Omron CX-Programmer project NuovoProgetto (CX-Programmer 8.01)

# PLC PLC: CJ1M CPU23

## Global symbols (name address type ; comment)
A W5 INT  ; PER AZZERAMENTO VARIABILI
A0.01 BOOL  ; 0.2
CICLO W0.00 BOOL[15]
CancelloAutomatico cancello_automatico
ControlloLivello controllo_livello
ENABLE W0.15 BOOL
GARAGE garage
IN00 0.00 BOOL  ; IN00
IN01 0.01 BOOL  ; IN01
IN02 0.02 BOOL  ; IN02
IN03 0.03 BOOL  ; IN03
IN04 0.04 BOOL  ; IN04
IN05 0.05 BOOL  ; IN05
IN06 0.06 BOOL  ; IN06
IN07 0.07 BOOL  ; IN07
IN08 0.08 BOOL  ; IN08
IN09 0.09 BOOL  ; IN09
IN10 0.10 BOOL  ; IN10
IN11 0.11 BOOL  ; IN11
IN12 0.12 BOOL  ; IN12
IN13 0.13 BOOL  ; IN13
IN14 0.14 BOOL  ; IN14
IN15 0.15 BOOL  ; IN15
IN16 1.00 BOOL  ; IN16
MAT2 inversione_di_marcia_MAT
MAT3 stella_triangolo_MAT
MarciaArresto marcia_arresto_MAT
Miscelatore miscelatore
OLD_OPZIONE W10 INT
OPZIONE W15 INT  ; SCELTA DEL CICLO
OUT00 2.00 BOOL  ; OUT00
OUT01 2.01 BOOL  ; OUT01
OUT02 2.02 BOOL  ; OUT02
OUT03 2.03 BOOL  ; OUT03
OUT04 2.04 BOOL  ; OUT04
OUT05 2.05 BOOL  ; OUT05
OUT06 2.06 BOOL  ; OUT06
OUT07 2.07 BOOL  ; OUT07
OUT08 2.08 BOOL  ; OUT08
OUT09 2.09 BOOL  ; OUT09
OUT10 2.10 BOOL  ; OUT10
OUT11 2.11 BOOL  ; OUT11
OUT12 2.12 BOOL  ; OUT12
OUT13 2.13 BOOL  ; OUT13
OUT14 2.14 BOOL  ; OUT14
OUT15 2.15 BOOL  ; OUT15
OUTCOUNTER1 D60 INT  ; uscita visione counter1
OUTCOUNTER2 D70 INT  ; uscita visione counter2
OUTCOUNTER3 D80 INT  ; uscita visione counter3
OUTCOUNTER4 D90 INT  ; uscita visione counter4
OUTCOUNTER5 D100 INT  ; uscita visione counter5
OUTCOUNTER6 D110 INT  ; uscita visione counter6
OUTTIMER1 D0 INT  ; uscita visione timer1
OUTTIMER2 D10 INT  ; uscita visione timer2
OUTTIMER3 D20 INT  ; uscita visione timer3
OUTTIMER4 D30 INT  ; uscita visione timer4
OUTTIMER5 D40 INT  ; uscita visione timer5
OUTTIMER6 D50 INT  ; uscita visione timer6
START 0.08 BOOL  ; INStart
SemaforoPedonale semaforo_pedonale
elp2 ciclo_elettropneumatico_due
elp3 ciclo_elettropneumatico_tre_mono
pos3 ciclo_elettropneumatico_uno

## Program CICLO_AVVIO (cyclic task 0)
; CICLO DI PARTENZA CON LA DEFINIZIONE DI TUTTI I BLOCCHI
Local symbols
RESET W100.02 BOOL
TERM1 W100.00 BOOL
TERM2 W100.01 BOOL

### Section RICHIAMMO_BLOCCHI

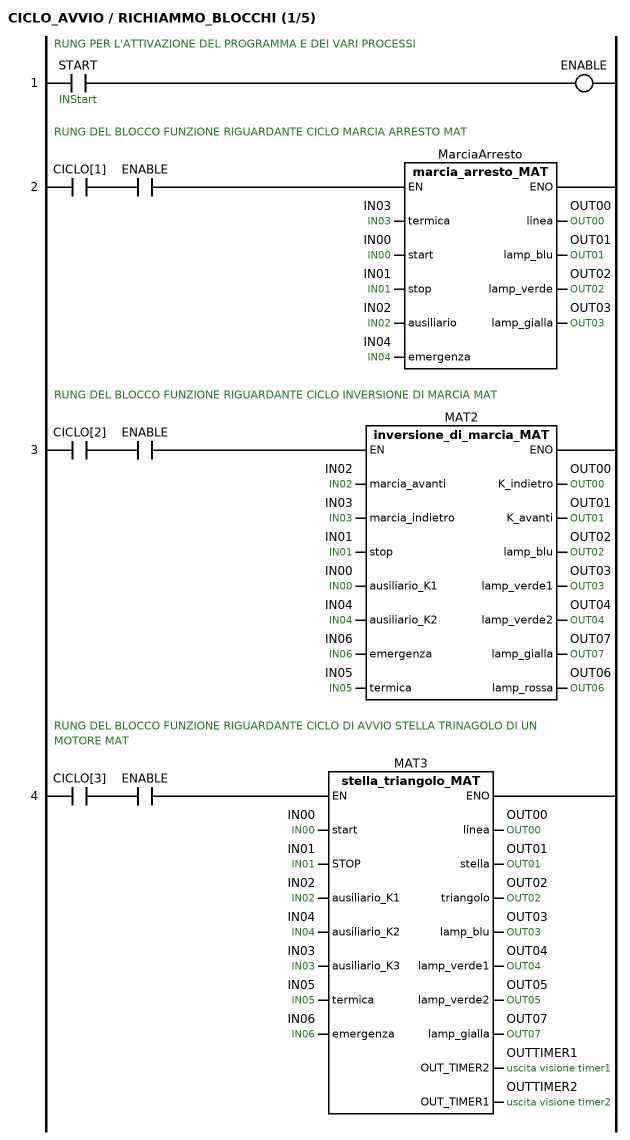
; rung 1: RUNG PER L'ATTIVAZIONE DEL PROGRAMMA E DEI VARI PROCESSI
LD START  ; INStart
OUT ENABLE
; rung 2: RUNG DEL BLOCCO FUNZIONE RIGUARDANTE CICLO MARCIA ARRESTO MAT
LD CICLO[1]
AND ENABLE
CALL MarciaArresto : marcia_arresto_MAT (termica := IN03, start := IN00, stop := IN01, ausiliario := IN02, emergenza := IN04, linea => OUT00, lamp_blu => OUT01, lamp_verde => OUT02, lamp_gialla => OUT03)  ; IN03, IN00, IN01, IN02, IN04, OUT00, OUT01, OUT02, OUT03
; rung 3: RUNG DEL BLOCCO FUNZIONE RIGUARDANTE CICLO INVERSIONE DI MARCIA MAT
LD CICLO[2]
AND ENABLE
CALL MAT2 : inversione_di_marcia_MAT (marcia_avanti := IN02, marcia_indietro := IN03, stop := IN01, ausiliario_K1 := IN00, ausiliario_K2 := IN04, emergenza := IN06, termica := IN05, K_indietro => OUT00, K_avanti => OUT01, lamp_blu => OUT02, lamp_verde1 => OUT03, lamp_verde2 => OUT04, lamp_gialla => OUT07, lamp_rossa => OUT06)  ; IN02, IN03, IN01, IN00, IN04, IN06, IN05, OUT00, OUT01, OUT02, OUT03, OUT04, OUT07, OUT06
; rung 4: RUNG DEL BLOCCO FUNZIONE RIGUARDANTE CICLO DI AVVIO STELLA TRINAGOLO DI UN MOTORE MAT
LD CICLO[3]
AND ENABLE
CALL MAT3 : stella_triangolo_MAT (start := IN00, STOP := IN01, ausiliario_K1 := IN02, ausiliario_K2 := IN04, ausiliario_K3 := IN03, termica := IN05, emergenza := IN06, linea => OUT00, stella => OUT01, triangolo => OUT02, lamp_blu => OUT03, lamp_verde1 => OUT04, lamp_verde2 => OUT05, lamp_gialla => OUT07, OUT_TIMER2 => OUTTIMER1, OUT_TIMER1 => OUTTIMER2)  ; IN00, IN01, IN02, IN04, IN03, IN05, IN06, OUT00, OUT01, OUT02, OUT03, OUT04, OUT05, OUT07, uscita visione timer1, uscita visione timer2

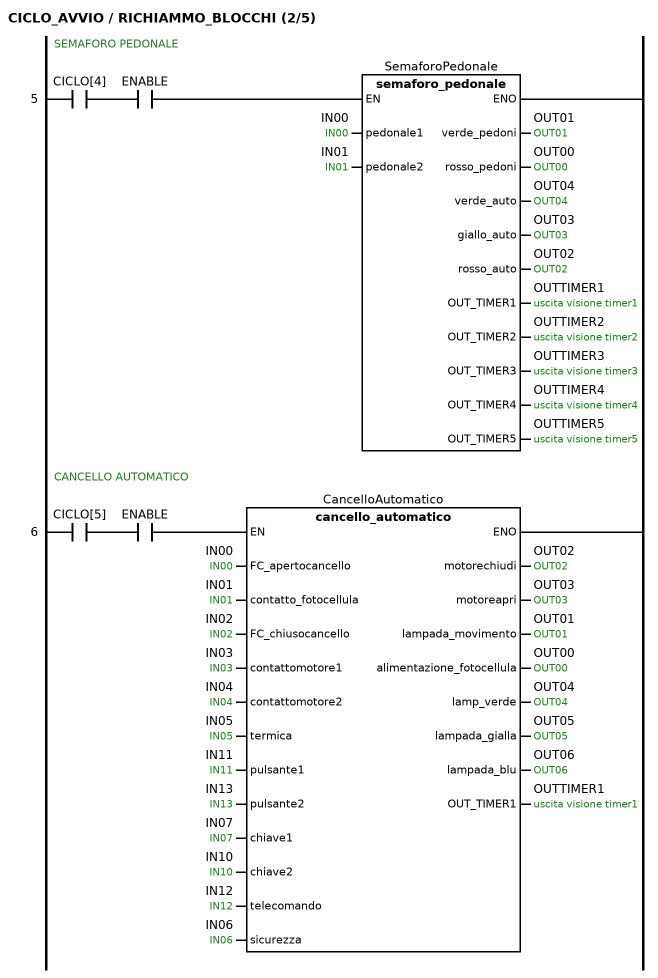
; rung 5: SEMAFORO PEDONALE
LD CICLO[4]
AND ENABLE
CALL SemaforoPedonale : semaforo_pedonale (pedonale1 := IN00, pedonale2 := IN01, verde_pedoni => OUT01, rosso_pedoni => OUT00, verde_auto => OUT04, giallo_auto => OUT03, rosso_auto => OUT02, OUT_TIMER1 => OUTTIMER1, OUT_TIMER2 => OUTTIMER2, OUT_TIMER3 => OUTTIMER3, OUT_TIMER4 => OUTTIMER4, OUT_TIMER5 => OUTTIMER5)  ; IN00, IN01, OUT01, OUT00, OUT04, OUT03, OUT02, uscita visione timer1, uscita visione timer2, uscita visione timer3, uscita visione timer4, uscita visione timer5
; rung 6: CANCELLO AUTOMATICO
LD CICLO[5]
AND ENABLE
CALL CancelloAutomatico : cancello_automatico (FC_apertocancello := IN00, contatto_fotocellula := IN01, FC_chiusocancello := IN02, contattomotore1 := IN03, contattomotore2 := IN04, termica := IN05, pulsante1 := IN11, pulsante2 := IN13, chiave1 := IN07, chiave2 := IN10, telecomando := IN12, sicurezza := IN06, motorechiudi => OUT02, motoreapri => OUT03, lampada_movimento => OUT01, alimentazione_fotocellula => OUT00, lamp_verde => OUT04, lampada_gialla => OUT05, lampada_blu => OUT06, OUT_TIMER1 => OUTTIMER1)  ; IN00, IN01, IN02, IN03, IN04, IN05, IN11, IN13, IN07, IN10, IN12, IN06, OUT02, OUT03, OUT01, OUT00, OUT04, OUT05, OUT06, uscita visione timer1

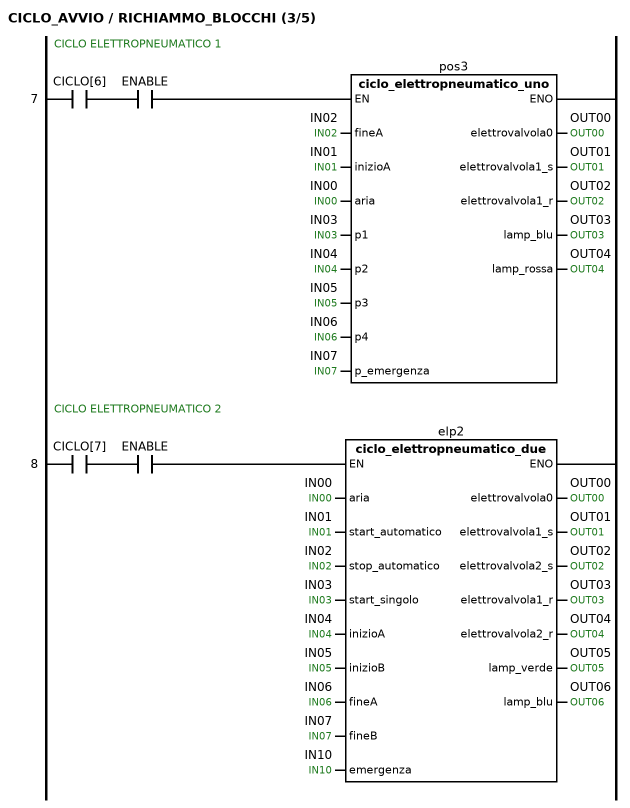
; rung 7: CICLO ELETTROPNEUMATICO 1
LD CICLO[6]
AND ENABLE
CALL pos3 : ciclo_elettropneumatico_uno (fineA := IN02, inizioA := IN01, aria := IN00, p1 := IN03, p2 := IN04, p3 := IN05, p4 := IN06, p_emergenza := IN07, elettrovalvola0 => OUT00, elettrovalvola1_s => OUT01, elettrovalvola1_r => OUT02, lamp_blu => OUT03, lamp_rossa => OUT04)  ; IN02, IN01, IN00, IN03, IN04, IN05, IN06, IN07, OUT00, OUT01, OUT02, OUT03, OUT04
; rung 8: CICLO ELETTROPNEUMATICO 2
LD CICLO[7]
AND ENABLE
CALL elp2 : ciclo_elettropneumatico_due (aria := IN00, start_automatico := IN01, stop_automatico := IN02, start_singolo := IN03, inizioA := IN04, inizioB := IN05, fineA := IN06, fineB := IN07, emergenza := IN10, elettrovalvola0 => OUT00, elettrovalvola1_s => OUT01, elettrovalvola2_s => OUT02, elettrovalvola1_r => OUT03, elettrovalvola2_r => OUT04, lamp_verde => OUT05, lamp_blu => OUT06)  ; IN00, IN01, IN02, IN03, IN04, IN05, IN06, IN07, IN10, OUT00, OUT01, OUT02, OUT03, OUT04, OUT05, OUT06

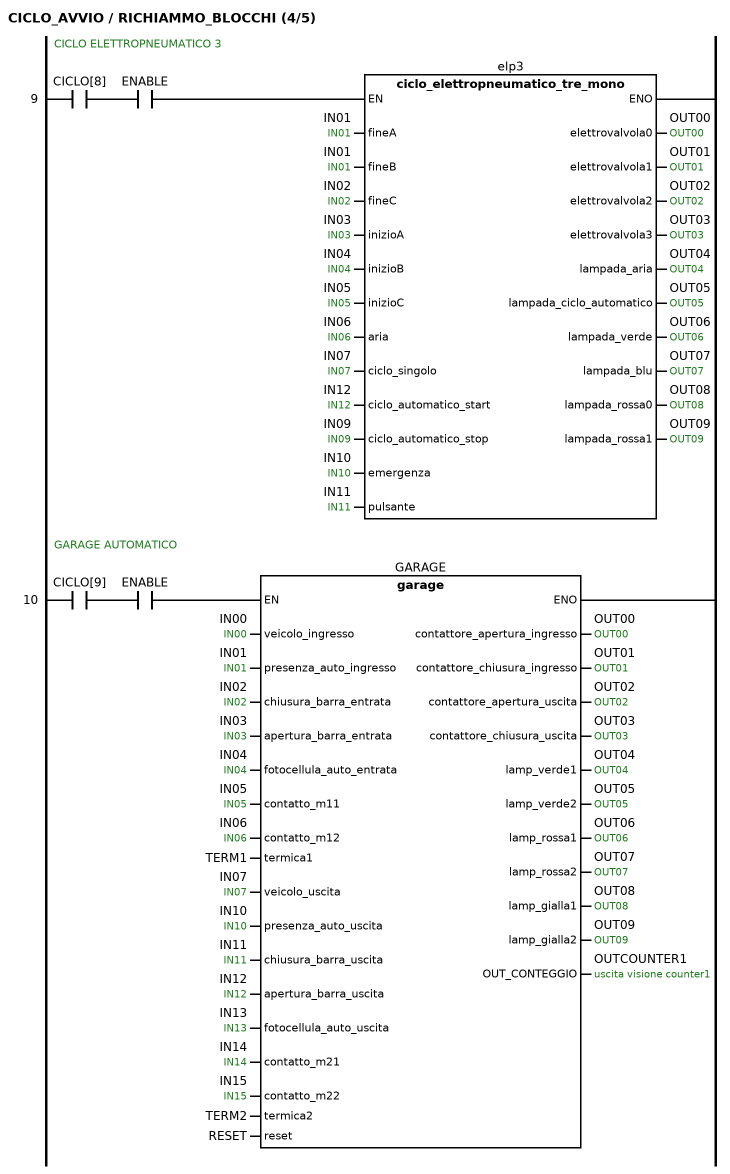
; rung 9: CICLO ELETTROPNEUMATICO 3
LD CICLO[8]
AND ENABLE
CALL elp3 : ciclo_elettropneumatico_tre_mono (fineA := IN01, fineB := IN01, fineC := IN02, inizioA := IN03, inizioB := IN04, inizioC := IN05, aria := IN06, ciclo_singolo := IN07, ciclo_automatico_start := IN12, ciclo_automatico_stop := IN09, emergenza := IN10, pulsante := IN11, elettrovalvola0 => OUT00, elettrovalvola1 => OUT01, elettrovalvola2 => OUT02, elettrovalvola3 => OUT03, lampada_aria => OUT04, lampada_ciclo_automatico => OUT05, lampada_verde => OUT06, lampada_blu => OUT07, lampada_rossa0 => OUT08, lampada_rossa1 => OUT09)  ; IN01, IN02, IN03, IN04, IN05, IN06, IN07, IN12, IN09, IN10, IN11, OUT00, OUT01, OUT02, OUT03, OUT04, OUT05, OUT06, OUT07, OUT08, OUT09
; rung 10: GARAGE AUTOMATICO
LD CICLO[9]
AND ENABLE
CALL GARAGE : garage (veicolo_ingresso := IN00, presenza_auto_ingresso := IN01, chiusura_barra_entrata := IN02, apertura_barra_entrata := IN03, fotocellula_auto_entrata := IN04, contatto_m11 := IN05, contatto_m12 := IN06, termica1 := TERM1, veicolo_uscita := IN07, presenza_auto_uscita := IN10, chiusura_barra_uscita := IN11, apertura_barra_uscita := IN12, fotocellula_auto_uscita := IN13, contatto_m21 := IN14, contatto_m22 := IN15, termica2 := TERM2, reset := RESET, contattore_apertura_ingresso => OUT00, contattore_chiusura_ingresso => OUT01, contattore_apertura_uscita => OUT02, contattore_chiusura_uscita => OUT03, lamp_verde1 => OUT04, lamp_verde2 => OUT05, lamp_rossa1 => OUT06, lamp_rossa2 => OUT07, lamp_gialla1 => OUT08, lamp_gialla2 => OUT09, OUT_CONTEGGIO => OUTCOUNTER1)  ; IN00, IN01, IN02, IN03, IN04, IN05, IN06, IN07, IN10, IN11, IN12, IN13, IN14, IN15, OUT00, OUT01, OUT02, OUT03, OUT04, OUT05, OUT06, OUT07, OUT08, OUT09, uscita visione counter1

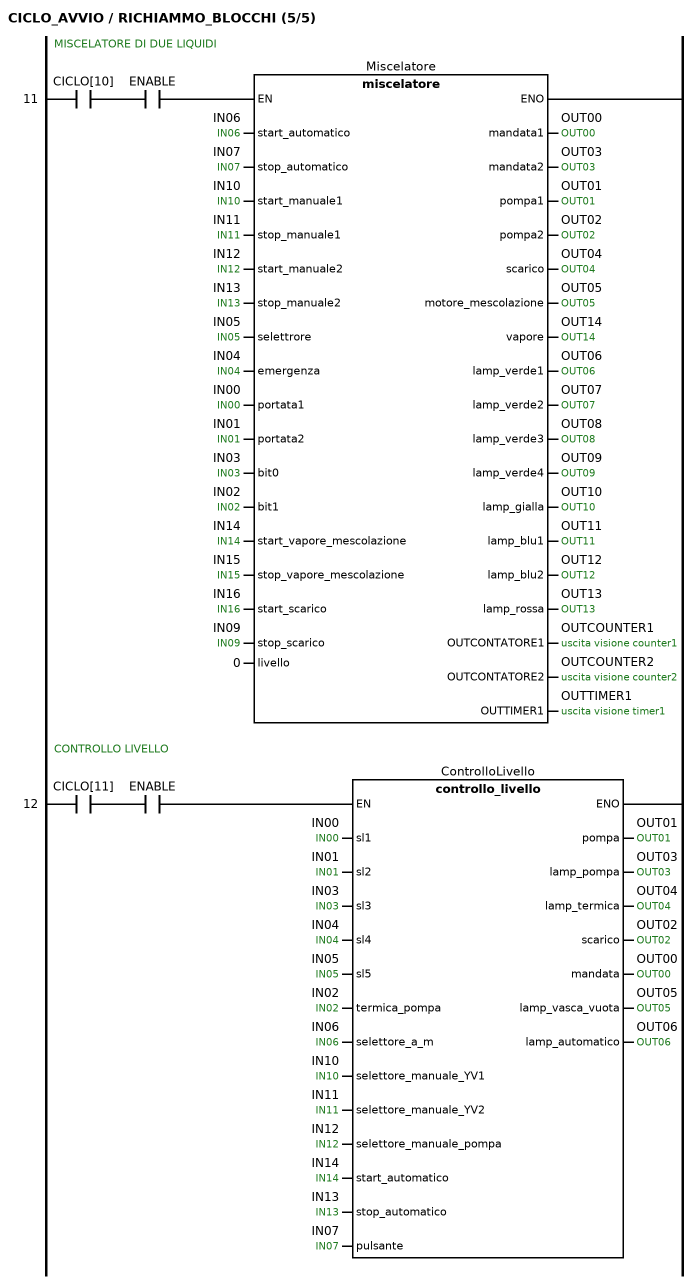
; rung 11: MISCELATORE DI DUE LIQUIDI
LD CICLO[10]
AND ENABLE
CALL Miscelatore : miscelatore (start_automatico := IN06, stop_automatico := IN07, start_manuale1 := IN10, stop_manuale1 := IN11, start_manuale2 := IN12, stop_manuale2 := IN13, selettrore := IN05, emergenza := IN04, portata1 := IN00, portata2 := IN01, bit0 := IN03, bit1 := IN02, start_vapore_mescolazione := IN14, stop_vapore_mescolazione := IN15, start_scarico := IN16, stop_scarico := IN09, livello := 0, mandata1 => OUT00, mandata2 => OUT03, pompa1 => OUT01, pompa2 => OUT02, scarico => OUT04, motore_mescolazione => OUT05, vapore => OUT14, lamp_verde1 => OUT06, lamp_verde2 => OUT07, lamp_verde3 => OUT08, lamp_verde4 => OUT09, lamp_gialla => OUT10, lamp_blu1 => OUT11, lamp_blu2 => OUT12, lamp_rossa => OUT13, OUTCONTATORE1 => OUTCOUNTER1, OUTCONTATORE2 => OUTCOUNTER2, OUTTIMER1 => OUTTIMER1)  ; IN06, IN07, IN10, IN11, IN12, IN13, IN05, IN04, IN00, IN01, IN03, IN02, IN14, IN15, IN16, IN09, OUT00, OUT03, OUT01, OUT02, OUT04, OUT05, OUT14, OUT06, OUT07, OUT08, OUT09, OUT10, OUT11, OUT12, OUT13, uscita visione counter1, uscita visione counter2, uscita visione timer1
; rung 12: CONTROLLO LIVELLO
LD CICLO[11]
AND ENABLE
CALL ControlloLivello : controllo_livello (sl1 := IN00, sl2 := IN01, sl3 := IN03, sl4 := IN04, sl5 := IN05, termica_pompa := IN02, selettore_a_m := IN06, selettore_manuale_YV1 := IN10, selettore_manuale_YV2 := IN11, selettore_manuale_pompa := IN12, start_automatico := IN14, stop_automatico := IN13, pulsante := IN07, pompa => OUT01, lamp_pompa => OUT03, lamp_termica => OUT04, scarico => OUT02, mandata => OUT00, lamp_vasca_vuota => OUT05, lamp_automatico => OUT06)  ; IN00, IN01, IN03, IN04, IN05, IN02, IN06, IN10, IN11, IN12, IN14, IN13, IN07, OUT01, OUT03, OUT04, OUT02, OUT00, OUT05, OUT06

### Section END
; rung 0
END(001)

## Program SCELTA (cyclic task 1)
; SCELTA
(*DOPO AVER RICEVUTO IL VALORE DI POSIZIONE SI ESEGUE LA VERIFICA COMPARANDO I VALORI PRECENTI  
CON QUELLI ATTUALI:
-SE CORRISPONDONO TUTTO OK  
-SE  DIVERSI VENGONO AGGIORNATI AI VALORI ATTUALI ( CICLO[] ) 
SUCCESSIVAMENTE MODIFICANO GLI ENABLE DEI BLOCCHI*)
IF ENABLE THEN
	
	IF OPZIONE =  OLD_OPZIONE THEN  		(* SE LA VARIABILE OPZIONE NON E' CAMBIATA NON ESEGUO NIENTE *)
	
			OLD_OPZIONE := OPZIONE;	
			
	ELSE
			(* AZZERAMENTO USCITE NEL CAMBIO DI STATO*)
			OUT00 := FALSE;
			OUT01 := FALSE;
			OUT02 := FALSE;
			OUT03 := FALSE;
			OUT04 := FALSE;
			OUT05 := FALSE;
			OUT06 := FALSE;
			OUT07 := FALSE;
			OUT08 := FALSE;
			OUT09 := FALSE;
			OUT10 := FALSE;
			OUT11 := FALSE;
			OUT12 := FALSE;
			OUT13 := FALSE;
			OUT14 := FALSE;
			OUT15:= FALSE;
			
			(* AZZERAMENTO USCITE NEL CAMBIO DI STATO*)			
			IN00 := FALSE;
			IN01 := FALSE;
			IN02 := FALSE;
			IN03 := FALSE;
			IN04 := FALSE;
			IN05 := FALSE;
			IN06 := FALSE;
			IN07 := FALSE;
			IN10 := FALSE;
			IN11 := FALSE;
			IN12 := FALSE;
			IN13 := FALSE;
			IN14 := FALSE;
			IN15:= FALSE;
			IN16 := FALSE;
				
                        (*SE LA VARIABILE OPZIONE E' CAMBIATA SI VERIFICA IL VALORE E SI CAMBIA IL BIT CORRISPONDENTE *)
			FOR A := 1 TO 11 BY 1 DO			(*CICLO PER ANDARE A CAMBIARE I VALORI DEI BIT*)

				IF A = OPZIONE  THEN            		(*CONFRONTO TRA INDICE E POSIZIONE*)
			
					CICLO[OPZIONE] := TRUE; 	(*SE IL VALORE E' UGUALE METTO A 1 IL BIT *)  
			
				ELSE
			
					CICLO[A] := FALSE; 		(*SE IL VALORE E' DIVERSO METTO A 0 IL BIT *)
			
				END_IF;
			
			END_FOR	;
	
	OLD_OPZIONE := OPZIONE; 			(*AGGIORNO IL VALORE DI OLD_OPZIONE*)

	END_IF;		

END_IF;;

## Function block cancello_automatico
VAR_INPUT
  FC_apertocancello : BOOL;
  contatto_fotocellula : BOOL;
  FC_chiusocancello : BOOL;
  contattomotore1 : BOOL;
  contattomotore2 : BOOL;
  termica : BOOL;
  pulsante1 : BOOL;
  pulsante2 : BOOL;
  chiave1 : BOOL;
  chiave2 : BOOL;
  telecomando : BOOL;
  sicurezza : BOOL;
END_VAR
VAR_OUTPUT
  motorechiudi : BOOL;
  motoreapri : BOOL;
  lampada_movimento : BOOL;
  alimentazione_fotocellula : BOOL;
  lamp_verde : BOOL;
  lampada_gialla : BOOL;
  lampada_blu : BOOL;
  OUT_TIMER1 : INT;
END_VAR
VAR
  MEM1 : BOOL;
  MEM2 : BOOL;
  MEM3 : BOOL;
  TIME1 : TIMER;
END_VAR

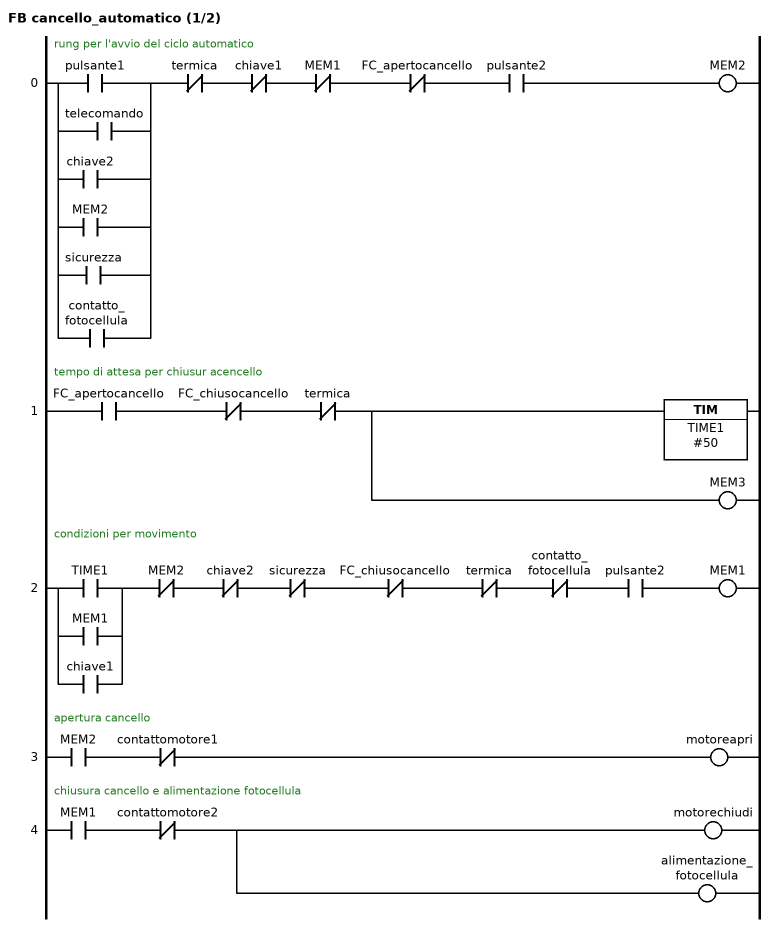
; rung 0: rung per l'avvio del ciclo automatico
LD pulsante1
OR telecomando
OR chiave2
OR MEM2
OR sicurezza
OR contatto_fotocellula
ANDNOT termica
ANDNOT chiave1
ANDNOT MEM1
ANDNOT FC_apertocancello
AND pulsante2
OUT MEM2
; rung 1: tempo di attesa per chiusur acencello
LD FC_apertocancello
ANDNOT FC_chiusocancello
ANDNOT termica
TIM TIME1 #50
OUT MEM3
; rung 2: condizioni per movimento
LD TIME1
OR MEM1
OR chiave1
ANDNOT MEM2
ANDNOT chiave2
ANDNOT sicurezza
ANDNOT FC_chiusocancello
ANDNOT termica
ANDNOT contatto_fotocellula
AND pulsante2
OUT MEM1
; rung 3: apertura cancello
LD MEM2
ANDNOT contattomotore1
OUT motoreapri
; rung 4: chiusura cancello e alimentazione fotocellula
LD MEM1
ANDNOT contattomotore2
OUT motorechiudi
OUT alimentazione_fotocellula

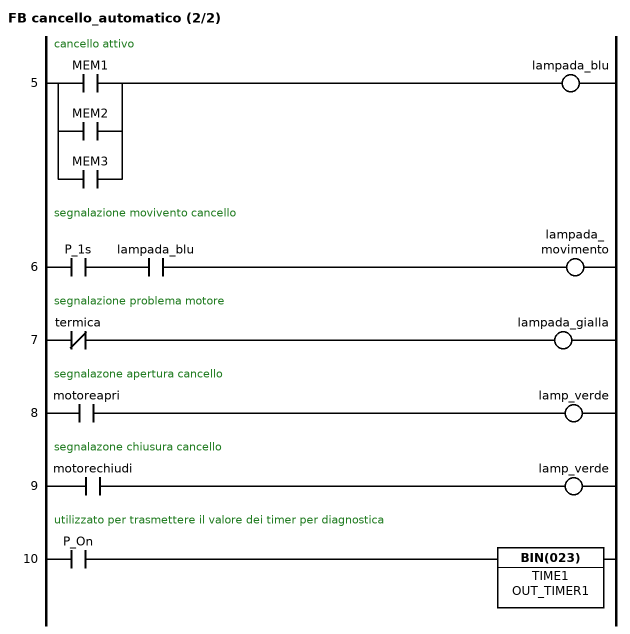
; rung 5: cancello attivo
LD MEM1
OR MEM2
OR MEM3
OUT lampada_blu
; rung 6: segnalazione movivento cancello
LD P_1s
AND lampada_blu
OUT lampada_movimento
; rung 7: segnalazione problema motore
LDNOT termica
OUT lampada_gialla
; rung 8: segnalazone apertura cancello
LD motoreapri
OUT lamp_verde
; rung 9: segnalazone chiusura cancello
LD motorechiudi
OUT lamp_verde
; rung 10: utilizzato per trasmettere il valore dei timer per diagnostica
LD P_On
BIN(023) TIME1 OUT_TIMER1

## Function block ciclo_elettropneumatico_due
VAR_INPUT
  aria : BOOL;
  start_automatico : BOOL;
  stop_automatico : BOOL;
  start_singolo : BOOL;
  inizioA : BOOL;
  inizioB : BOOL;
  fineA : BOOL;
  fineB : BOOL;
  emergenza : BOOL;
END_VAR
VAR_OUTPUT
  elettrovalvola0 : BOOL;
  elettrovalvola1_s : BOOL;
  elettrovalvola2_s : BOOL;
  elettrovalvola1_r : BOOL;
  elettrovalvola2_r : BOOL;
  lamp_verde : BOOL;
  lamp_blu : BOOL;
END_VAR
VAR
  MEM2 : BOOL;
  MEM1 : BOOL;
END_VAR

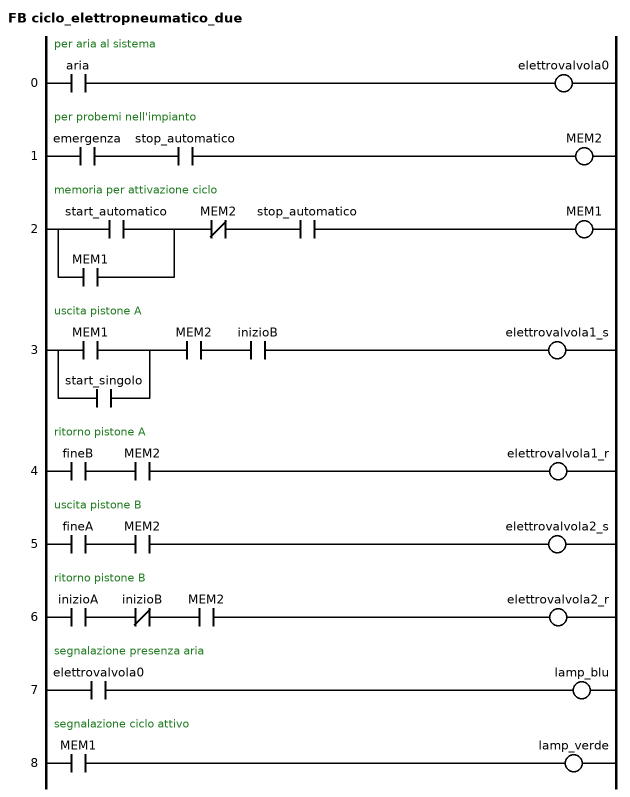
; rung 0: per aria al sistema
LD aria
OUT elettrovalvola0
; rung 1: per probemi nell'impianto
LD emergenza
AND stop_automatico
OUT MEM2
; rung 2: memoria per attivazione ciclo
LD start_automatico
OR MEM1
ANDNOT MEM2
AND stop_automatico
OUT MEM1
; rung 3: uscita pistone A
LD MEM1
OR start_singolo
AND MEM2
AND inizioB
OUT elettrovalvola1_s
; rung 4: ritorno pistone A
LD fineB
AND MEM2
OUT elettrovalvola1_r
; rung 5: uscita pistone B
LD fineA
AND MEM2
OUT elettrovalvola2_s
; rung 6: ritorno pistone B
LD inizioA
ANDNOT inizioB
AND MEM2
OUT elettrovalvola2_r
; rung 7: segnalazione presenza aria
LD elettrovalvola0
OUT lamp_blu
; rung 8: segnalazione ciclo attivo
LD MEM1
OUT lamp_verde

## Function block ciclo_elettropneumatico_tre_mono
VAR_INPUT
  fineA : BOOL;
  fineB : BOOL;
  fineC : BOOL;
  inizioA : BOOL;
  inizioB : BOOL;
  inizioC : BOOL;
  aria : BOOL;
  ciclo_singolo : BOOL;
  ciclo_automatico_start : BOOL;
  ciclo_automatico_stop : BOOL;
  emergenza : BOOL;
  pulsante : BOOL;
END_VAR
VAR_OUTPUT
  elettrovalvola0 : BOOL;
  elettrovalvola1 : BOOL;
  elettrovalvola2 : BOOL;
  elettrovalvola3 : BOOL;
  lampada_aria : BOOL;
  lampada_ciclo_automatico : BOOL;
  lampada_verde : BOOL;
  lampada_blu : BOOL;
  lampada_rossa0 : BOOL;
  lampada_rossa1 : BOOL;
END_VAR
VAR
  MEM1 : BOOL;
  MEM2 : BOOL;
END_VAR

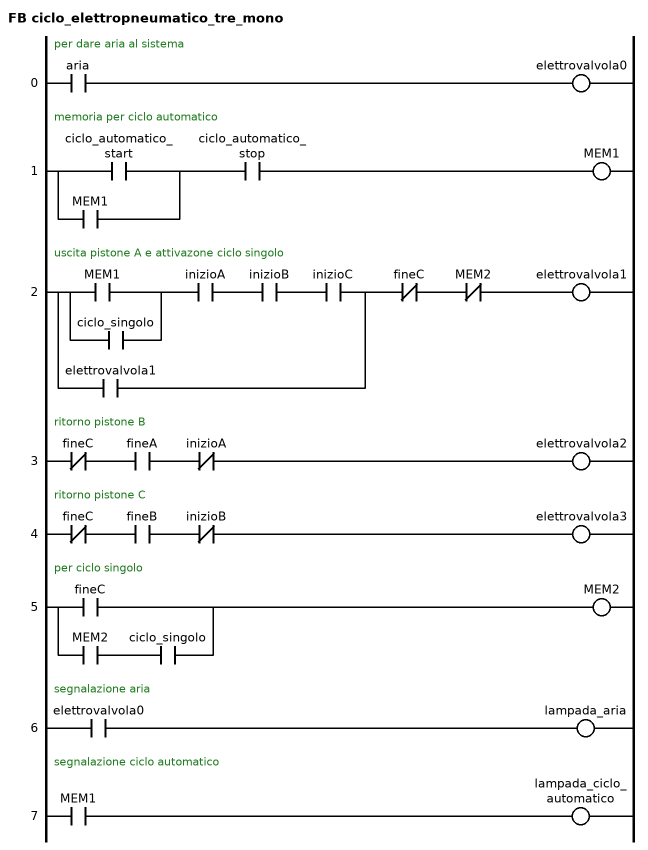
; rung 0: per dare aria al sistema
LD aria
OUT elettrovalvola0
; rung 1: memoria per ciclo automatico
LD ciclo_automatico_start
OR MEM1
AND ciclo_automatico_stop
OUT MEM1
; rung 2: uscita pistone A e attivazone ciclo singolo
LD MEM1
OR ciclo_singolo
AND inizioA
AND inizioB
AND inizioC
OR elettrovalvola1
ANDNOT fineC
ANDNOT MEM2
OUT elettrovalvola1
; rung 3: ritorno pistone B
LDNOT fineC
AND fineA
ANDNOT inizioA
OUT elettrovalvola2
; rung 4: ritorno pistone C
LDNOT fineC
AND fineB
ANDNOT inizioB
OUT elettrovalvola3
; rung 5: per ciclo singolo
LD fineC
LD MEM2
AND ciclo_singolo
ORLD
OUT MEM2
; rung 6: segnalazione aria
LD elettrovalvola0
OUT lampada_aria
; rung 7: segnalazione ciclo automatico
LD MEM1
OUT lampada_ciclo_automatico

## Function block ciclo_elettropneumatico_uno
VAR_INPUT
  fineA : BOOL;
  inizioA : BOOL;
  aria : BOOL;
  p1 : BOOL;
  p2 : BOOL;
  p3 : BOOL;
  p4 : BOOL;
  p_emergenza : BOOL;
END_VAR
VAR_OUTPUT
  elettrovalvola0 : BOOL;
  elettrovalvola1_s : BOOL;
  elettrovalvola1_r : BOOL;
  lamp_blu : BOOL;
  lamp_rossa : BOOL;
END_VAR
VAR
  MEM1 : BOOL;
  MEM2 : BOOL;
END_VAR

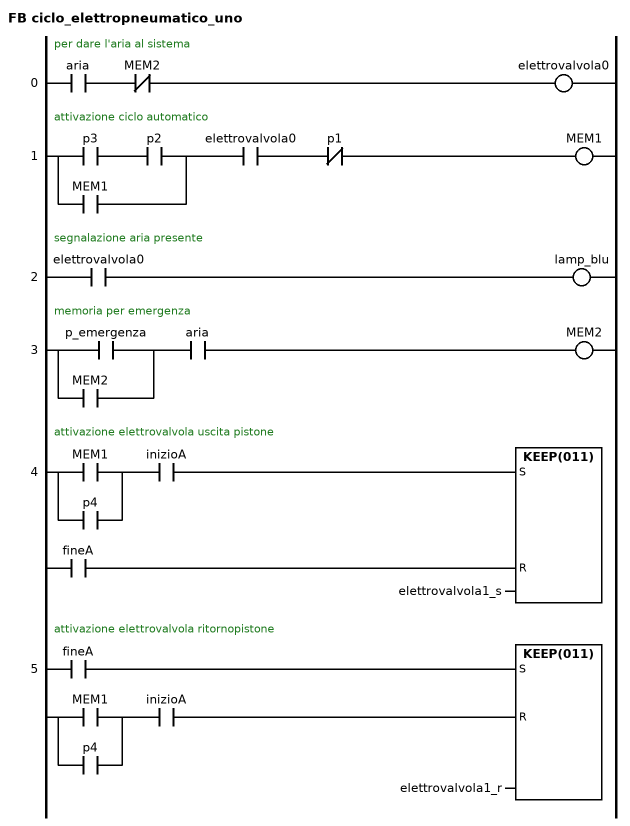
; rung 0: per dare l'aria al sistema
LD aria
ANDNOT MEM2
OUT elettrovalvola0
; rung 1: attivazione ciclo automatico
LD p3
AND p2
OR MEM1
AND elettrovalvola0
ANDNOT p1
OUT MEM1
; rung 2: segnalazione aria presente
LD elettrovalvola0
OUT lamp_blu
; rung 3: memoria per emergenza
LD p_emergenza
OR MEM2
AND aria
OUT MEM2
; rung 4: attivazione elettrovalvola uscita pistone
LD MEM1
OR p4
AND inizioA
LD fineA
KEEP(011) elettrovalvola1_s
; rung 5: attivazione elettrovalvola ritornopistone
LD fineA
LD MEM1
OR p4
AND inizioA
KEEP(011) elettrovalvola1_r

## Function block controllo_livello
VAR_INPUT
  sl1 : BOOL;
  sl2 : BOOL;
  sl3 : BOOL;
  sl4 : BOOL;
  sl5 : BOOL;
  termica_pompa : BOOL;
  selettore_a_m : BOOL;
  selettore_manuale_YV1 : BOOL;
  selettore_manuale_YV2 : BOOL;
  selettore_manuale_pompa : BOOL;
  start_automatico : BOOL;
  stop_automatico : BOOL;
  pulsante : BOOL;
END_VAR
VAR_OUTPUT
  pompa : BOOL;
  lamp_pompa : BOOL;
  lamp_termica : BOOL;
  scarico : BOOL;
  mandata : BOOL;
  lamp_vasca_vuota : BOOL;
  lamp_automatico : BOOL;
END_VAR
VAR
  MEM1 : BOOL;
  MEM2 : BOOL;
  MEM3 : BOOL;
  MEM4 : BOOL;
  MEM5 : BOOL;
  MEM6 : BOOL;
  MEM7 : BOOL;
  MEM8 : BOOL;
END_VAR

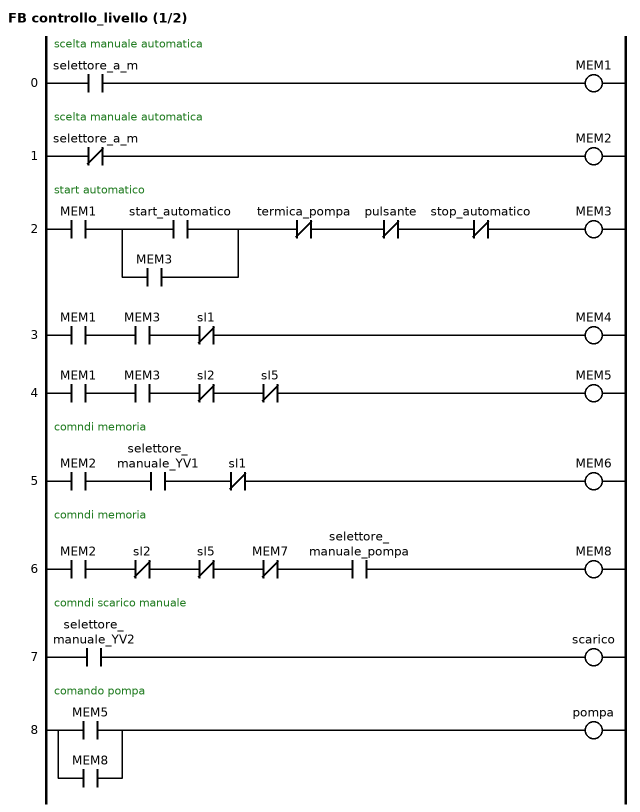
; rung 0: scelta manuale automatica
LD selettore_a_m
OUT MEM1
; rung 1: scelta manuale automatica
LDNOT selettore_a_m
OUT MEM2
; rung 2: start automatico
LD MEM1
LD start_automatico
OR MEM3
ANDLD
ANDNOT termica_pompa
ANDNOT pulsante
ANDNOT stop_automatico
OUT MEM3
; rung 3
LD MEM1
AND MEM3
ANDNOT sl1
OUT MEM4
; rung 4
LD MEM1
AND MEM3
ANDNOT sl2
ANDNOT sl5
OUT MEM5
; rung 5: comndi memoria
LD MEM2
AND selettore_manuale_YV1
ANDNOT sl1
OUT MEM6
; rung 6: comndi memoria
LD MEM2
ANDNOT sl2
ANDNOT sl5
ANDNOT MEM7
AND selettore_manuale_pompa
OUT MEM8
; rung 7: comndi scarico manuale
LD selettore_manuale_YV2
OUT scarico
; rung 8: comando pompa
LD MEM5
OR MEM8
OUT pompa

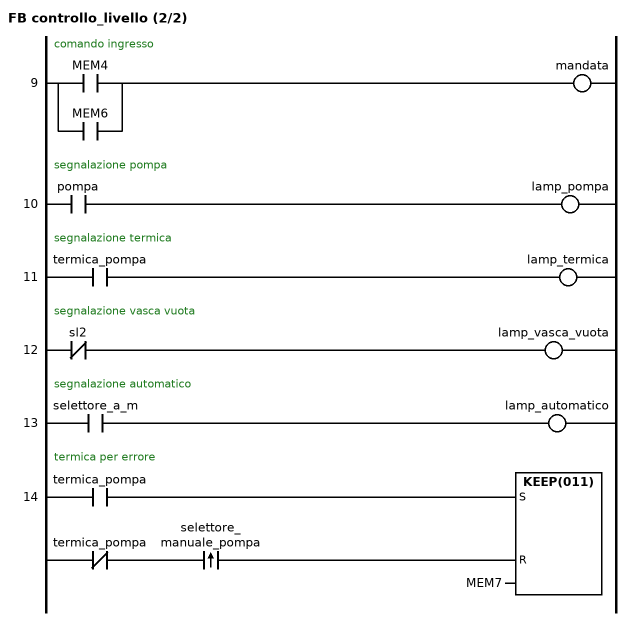
; rung 9: comando ingresso
LD MEM4
OR MEM6
OUT mandata
; rung 10: segnalazione pompa
LD pompa
OUT lamp_pompa
; rung 11: segnalazione termica
LD termica_pompa
OUT lamp_termica
; rung 12: segnalazione vasca vuota
LDNOT sl2
OUT lamp_vasca_vuota
; rung 13: segnalazione automatico
LD selettore_a_m
OUT lamp_automatico
; rung 14: termica per errore
LD termica_pompa
LDNOT termica_pompa
@AND selettore_manuale_pompa
KEEP(011) MEM7

## Function block garage
VAR_INPUT
  veicolo_ingresso : BOOL;
  presenza_auto_ingresso : BOOL;
  chiusura_barra_entrata : BOOL;
  apertura_barra_entrata : BOOL;
  fotocellula_auto_entrata : BOOL;
  contatto_m11 : BOOL;
  contatto_m12 : BOOL;
  termica1 : BOOL;
  veicolo_uscita : BOOL;
  presenza_auto_uscita : BOOL;
  chiusura_barra_uscita : BOOL;
  apertura_barra_uscita : BOOL;
  fotocellula_auto_uscita : BOOL;
  contatto_m21 : BOOL;
  contatto_m22 : BOOL;
  termica2 : BOOL;
  reset : BOOL;
END_VAR
VAR_OUTPUT
  contattore_apertura_ingresso : BOOL;
  contattore_chiusura_ingresso : BOOL;
  contattore_apertura_uscita : BOOL;
  contattore_chiusura_uscita : BOOL;
  lamp_verde1 : BOOL;
  lamp_verde2 : BOOL;
  lamp_rossa1 : BOOL;
  lamp_rossa2 : BOOL;
  lamp_gialla1 : BOOL;
  lamp_gialla2 : BOOL;
  OUT_CONTEGGIO : INT;
END_VAR
VAR
  MEM1 : BOOL;
  MEM2 : BOOL;
  CONTA : COUNTER;
END_VAR

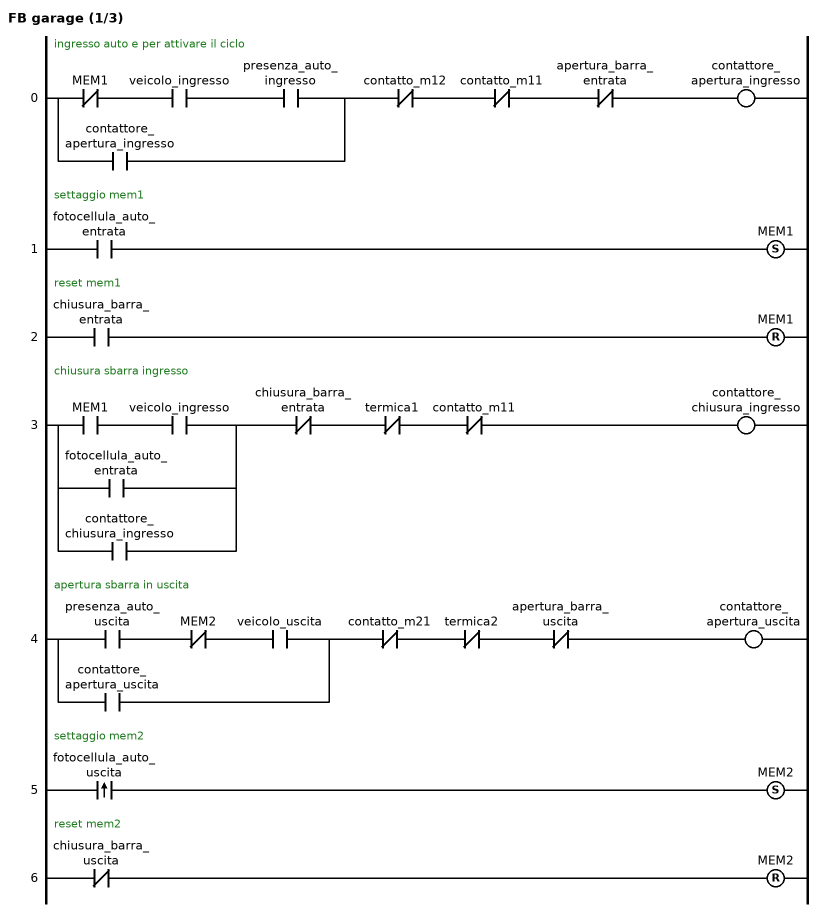
; rung 0: ingresso auto e per attivare il ciclo
LDNOT MEM1
AND veicolo_ingresso
AND presenza_auto_ingresso
OR contattore_apertura_ingresso
ANDNOT contatto_m12
ANDNOT contatto_m11
ANDNOT apertura_barra_entrata
OUT contattore_apertura_ingresso
; rung 1: settaggio mem1
LD fotocellula_auto_entrata
SET MEM1
; rung 2: reset mem1
LD chiusura_barra_entrata
RSET MEM1
; rung 3: chiusura sbarra ingresso
LD MEM1
AND veicolo_ingresso
OR fotocellula_auto_entrata
OR contattore_chiusura_ingresso
ANDNOT chiusura_barra_entrata
ANDNOT termica1
ANDNOT contatto_m11
OUT contattore_chiusura_ingresso
; rung 4: apertura sbarra in uscita
LD presenza_auto_uscita
ANDNOT MEM2
AND veicolo_uscita
OR contattore_apertura_uscita
ANDNOT contatto_m21
ANDNOT termica2
ANDNOT apertura_barra_uscita
OUT contattore_apertura_uscita
; rung 5: settaggio mem2
@LD fotocellula_auto_uscita
SET MEM2
; rung 6: reset mem2
LDNOT chiusura_barra_uscita
RSET MEM2

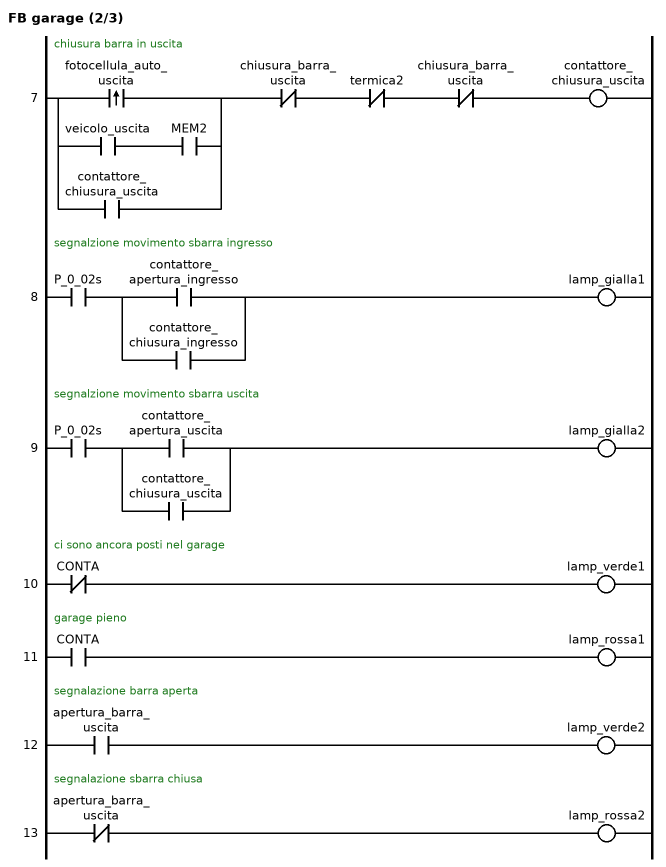
; rung 7: chiusura barra in uscita
@LD fotocellula_auto_uscita
LD veicolo_uscita
AND MEM2
ORLD
OR contattore_chiusura_uscita
ANDNOT chiusura_barra_uscita
ANDNOT termica2
ANDNOT chiusura_barra_uscita
OUT contattore_chiusura_uscita
; rung 8: segnalzione movimento sbarra ingresso
LD P_0_02s
LD contattore_apertura_ingresso
OR contattore_chiusura_ingresso
ANDLD
OUT lamp_gialla1
; rung 9: segnalzione movimento sbarra uscita
LD P_0_02s
LD contattore_apertura_uscita
OR contattore_chiusura_uscita
ANDLD
OUT lamp_gialla2
; rung 10: ci sono ancora posti nel garage
LDNOT CONTA
OUT lamp_verde1
; rung 11: garage pieno
LD CONTA
OUT lamp_rossa1
; rung 12: segnalazione barra aperta
LD apertura_barra_uscita
OUT lamp_verde2
; rung 13: segnalazione sbarra chiusa
LDNOT apertura_barra_uscita
OUT lamp_rossa2

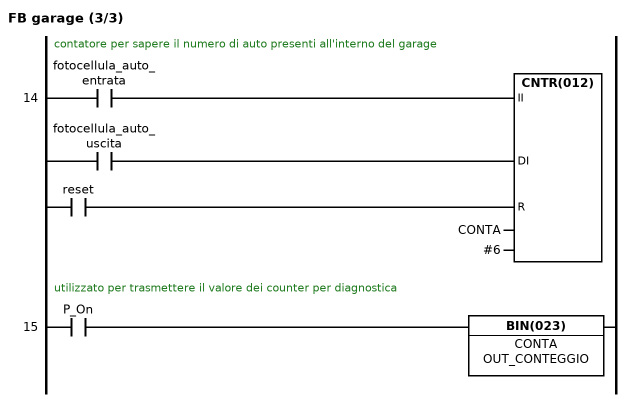
; rung 14: contatore per sapere il numero di auto presenti all'interno del garage
LD fotocellula_auto_entrata
LD fotocellula_auto_uscita
LD reset
CNTR(012) CONTA #6
; rung 15: utilizzato per trasmettere il valore dei counter per diagnostica
LD P_On
BIN(023) CONTA OUT_CONTEGGIO

## Function block inversione_di_marcia_MAT
VAR_INPUT
  marcia_avanti : BOOL;
  marcia_indietro : BOOL;
  stop : BOOL;
  ausiliario_K1 : BOOL;
  ausiliario_K2 : BOOL;
  emergenza : BOOL;
  termica : BOOL;
END_VAR
VAR_OUTPUT
  K_indietro : BOOL;
  K_avanti : BOOL;
  lamp_blu : BOOL;
  lamp_verde1 : BOOL;
  lamp_verde2 : BOOL;
  lamp_gialla : BOOL;
  lamp_rossa : BOOL;
END_VAR
VAR
  err : BOOL;
END_VAR

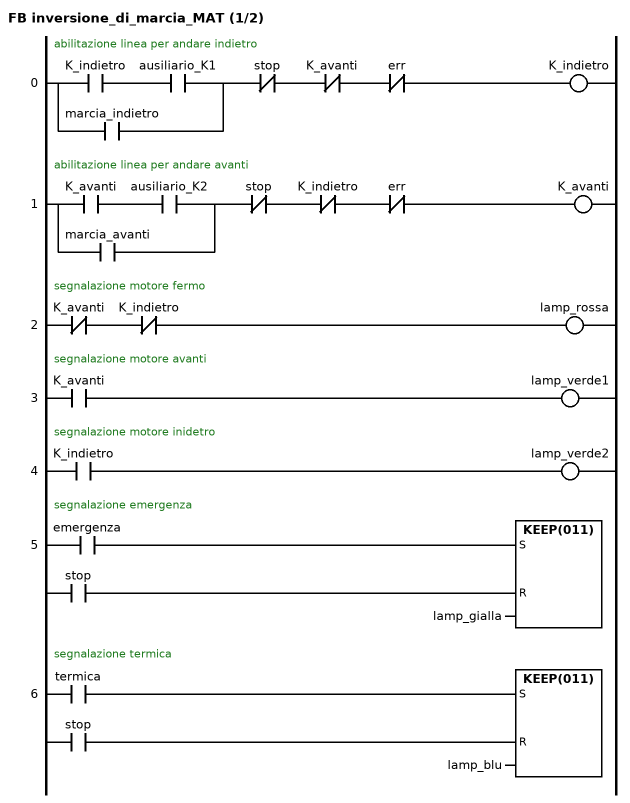
; rung 0: abilitazione linea per andare indietro
LD K_indietro
AND ausiliario_K1
OR marcia_indietro
ANDNOT stop
ANDNOT K_avanti
ANDNOT err
OUT K_indietro
; rung 1: abilitazione linea per andare avanti
LD K_avanti
AND ausiliario_K2
OR marcia_avanti
ANDNOT stop
ANDNOT K_indietro
ANDNOT err
OUT K_avanti
; rung 2: segnalazione motore fermo
LDNOT K_avanti
ANDNOT K_indietro
OUT lamp_rossa
; rung 3: segnalazione motore avanti
LD K_avanti
OUT lamp_verde1
; rung 4: segnalazione motore inidetro
LD K_indietro
OUT lamp_verde2
; rung 5: segnalazione emergenza
LD emergenza
LD stop
KEEP(011) lamp_gialla
; rung 6: segnalazione termica
LD termica
LD stop
KEEP(011) lamp_blu

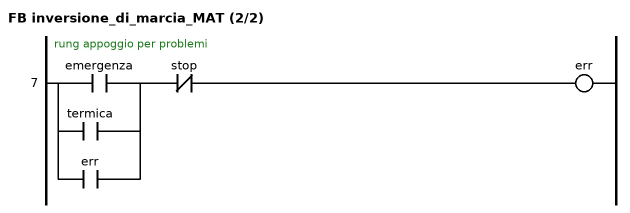
; rung 7: rung appoggio per problemi
LD emergenza
OR termica
OR err
ANDNOT stop
OUT err

## Function block marcia_arresto_MAT
VAR_INPUT
  termica : BOOL;
  start : BOOL;
  stop : BOOL;
  ausiliario : BOOL;
  emergenza : BOOL;
END_VAR
VAR_OUTPUT
  linea : BOOL;
  lamp_blu : BOOL;
  lamp_verde : BOOL;
  lamp_gialla : BOOL;
END_VAR
VAR
  err : BOOL;
END_VAR

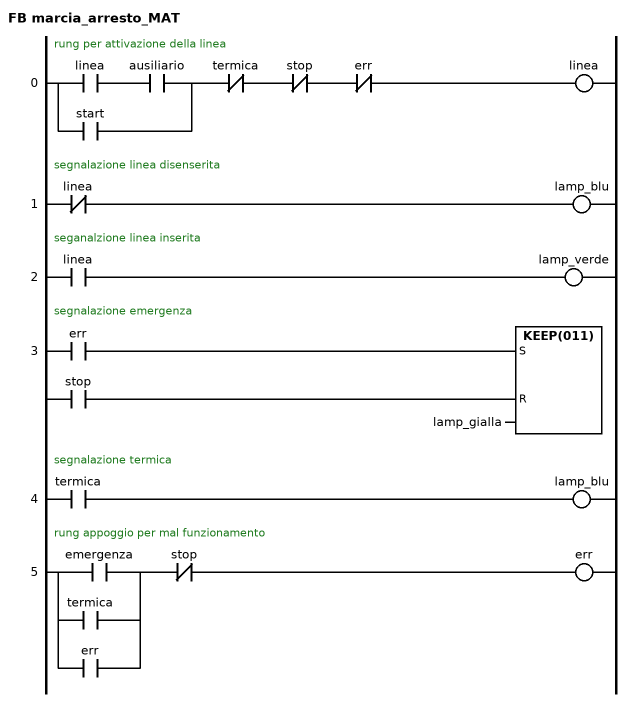
; rung 0: rung per attivazione della linea
LD linea
AND ausiliario
OR start
ANDNOT termica
ANDNOT stop
ANDNOT err
OUT linea
; rung 1: segnalazione linea disenserita
LDNOT linea
OUT lamp_blu
; rung 2: seganalzione linea inserita
LD linea
OUT lamp_verde
; rung 3: segnalazione emergenza
LD err
LD stop
KEEP(011) lamp_gialla
; rung 4: segnalazione termica
LD termica
OUT lamp_blu
; rung 5: rung appoggio per mal funzionamento
LD emergenza
OR termica
OR err
ANDNOT stop
OUT err

## Function block miscelatore
VAR_INPUT
  start_automatico : BOOL;
  stop_automatico : BOOL;
  start_manuale1 : BOOL;
  stop_manuale1 : BOOL;
  start_manuale2 : BOOL;
  stop_manuale2 : BOOL;
  selettrore : BOOL;
  emergenza : BOOL;
  portata1 : BOOL;
  portata2 : BOOL;
  bit0 : BOOL;
  bit1 : BOOL;
  start_vapore_mescolazione : BOOL;
  stop_vapore_mescolazione : BOOL;
  start_scarico : BOOL;
  stop_scarico : BOOL;
  livello : INT;
END_VAR
VAR_OUTPUT
  mandata1 : BOOL;  (* elettrovalvola *)
  mandata2 : BOOL;  (* elettrovalvola *)
  pompa1 : BOOL;
  pompa2 : BOOL;
  scarico : BOOL;  (* elettrovalvola *)
  motore_mescolazione : BOOL;
  vapore : BOOL;  (* elettrovalvola *)
  lamp_verde1 : BOOL;
  lamp_verde2 : BOOL;
  lamp_verde3 : BOOL;
  lamp_verde4 : BOOL;
  lamp_gialla : BOOL;
  lamp_blu1 : BOOL;
  lamp_blu2 : BOOL;
  lamp_rossa : BOOL;
  OUTCONTATORE1 : INT;
  OUTCONTATORE2 : INT;
  OUTTIMER1 : INT;
END_VAR
VAR
  MEM1 : BOOL;
  CONTA1 : COUNTER;
  CONTA2 : COUNTER;
  MEM2 : BOOL;
  MEM3 : BOOL;
  MEM4 : BOOL;
  TIMER : TIMER;
  MEM : BOOL;
  MEM5 : BOOL;  (* PER SCARICO *)
  MEM6 : BOOL;  (* MANUALE CARICO1 *)
  MEM7 : BOOL;  (* MANUALE CARICO 2 *)
  MEM8 : BOOL;  (* MANUALE VAPORE E MESCOLAZIONE *)
  ERR : BOOL;
  MEM10 : BOOL;
  MEM11 : BOOL;
  MEM12 : BOOL;
  MEM13 : BOOL;
  MEM14 : BOOL;
  MEM15 : BOOL;
  MEM20 : BOOL;
END_VAR

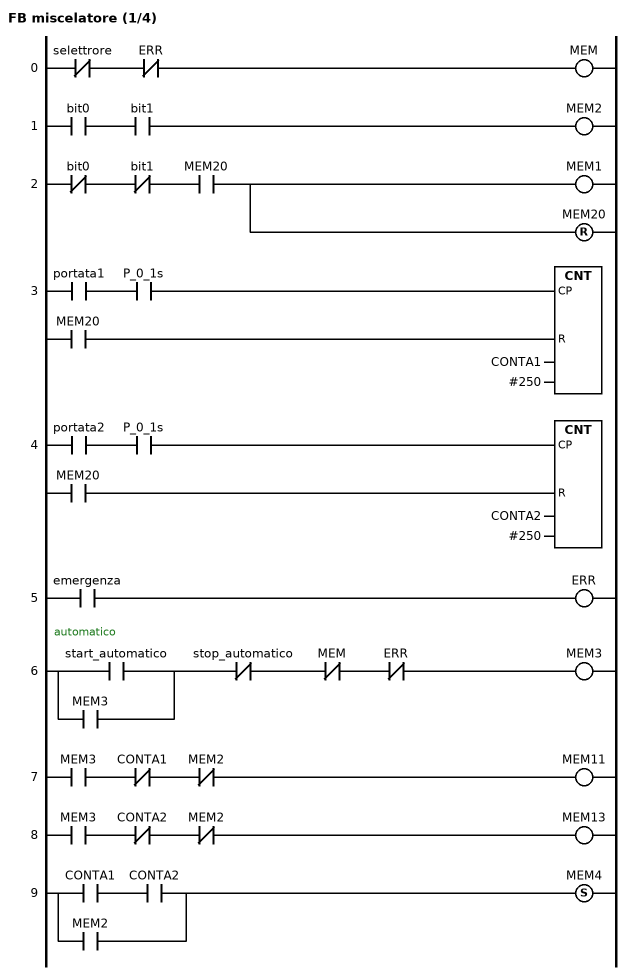
; rung 0
LDNOT selettrore
ANDNOT ERR
OUT MEM
; rung 1
LD bit0
AND bit1
OUT MEM2
; rung 2
LDNOT bit0
ANDNOT bit1
AND MEM20
OUT MEM1
RSET MEM20
; rung 3
LD portata1
AND P_0_1s
LD MEM20
CNT CONTA1 #250
; rung 4
LD portata2
AND P_0_1s
LD MEM20
CNT CONTA2 #250
; rung 5
LD emergenza
OUT ERR
; rung 6: automatico
LD start_automatico
OR MEM3
ANDNOT stop_automatico
ANDNOT MEM
ANDNOT ERR
OUT MEM3
; rung 7
LD MEM3
ANDNOT CONTA1
ANDNOT MEM2
OUT MEM11
; rung 8
LD MEM3
ANDNOT CONTA2
ANDNOT MEM2
OUT MEM13
; rung 9
LD CONTA1
AND CONTA2
OR MEM2
SET MEM4

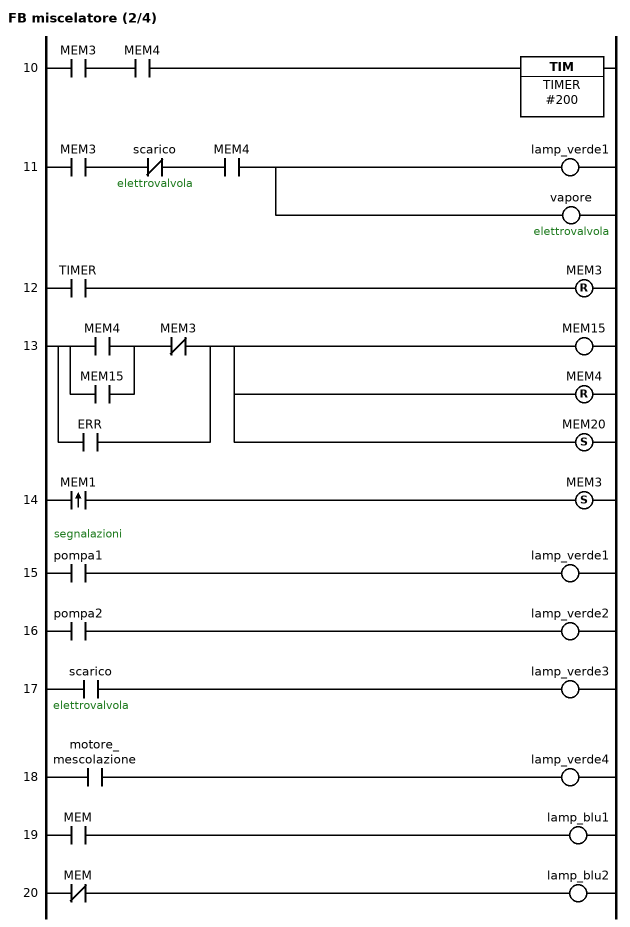
; rung 10
LD MEM3
AND MEM4
TIM TIMER #200
; rung 11
LD MEM3
ANDNOT scarico  ; elettrovalvola
AND MEM4
OUT lamp_verde1
OUT vapore  ; elettrovalvola
; rung 12
LD TIMER
RSET MEM3
; rung 13
LD MEM4
OR MEM15
ANDNOT MEM3
OR ERR
OUT MEM15
RSET MEM4
SET MEM20
; rung 14
@LD MEM1
SET MEM3
; rung 15: segnalazioni
LD pompa1
OUT lamp_verde1
; rung 16
LD pompa2
OUT lamp_verde2
; rung 17
LD scarico  ; elettrovalvola
OUT lamp_verde3
; rung 18
LD motore_mescolazione
OUT lamp_verde4
; rung 19
LD MEM
OUT lamp_blu1
; rung 20
LDNOT MEM
OUT lamp_blu2

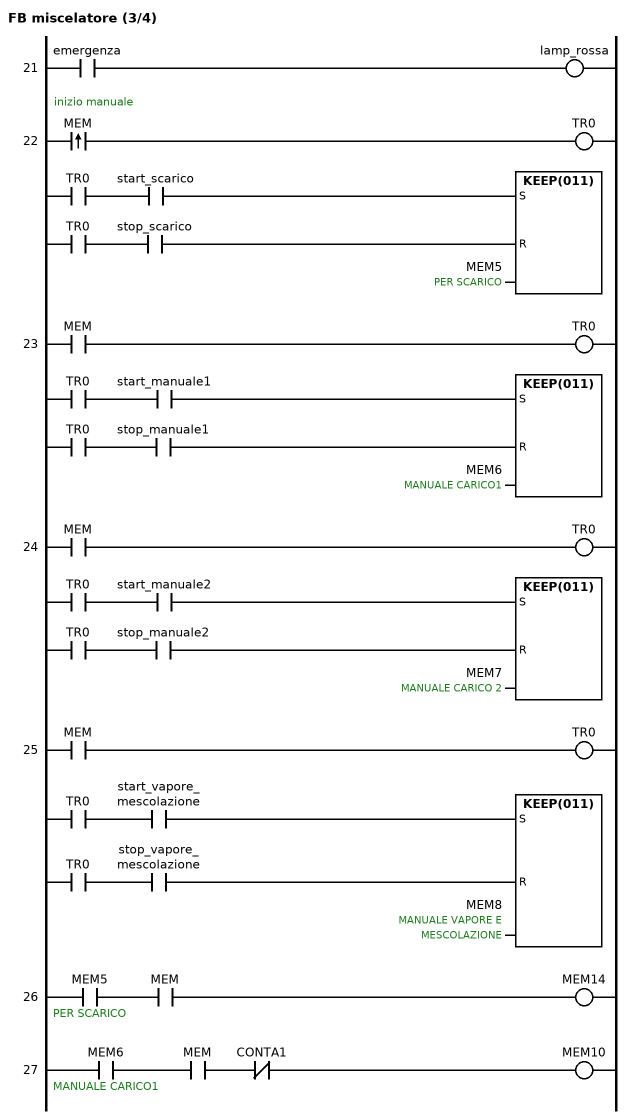
; rung 21
LD emergenza
OUT lamp_rossa
; rung 22: inizio manuale
@LD MEM
OUT TR0
LD TR0
AND start_scarico
LD TR0
AND stop_scarico
KEEP(011) MEM5  ; PER SCARICO
; rung 23
LD MEM
OUT TR0
LD TR0
AND start_manuale1
LD TR0
AND stop_manuale1
KEEP(011) MEM6  ; MANUALE CARICO1
; rung 24
LD MEM
OUT TR0
LD TR0
AND start_manuale2
LD TR0
AND stop_manuale2
KEEP(011) MEM7  ; MANUALE CARICO 2
; rung 25
LD MEM
OUT TR0
LD TR0
AND start_vapore_mescolazione
LD TR0
AND stop_vapore_mescolazione
KEEP(011) MEM8  ; MANUALE VAPORE E MESCOLAZIONE
; rung 26
LD MEM5  ; PER SCARICO
AND MEM
OUT MEM14
; rung 27
LD MEM6  ; MANUALE CARICO1
AND MEM
ANDNOT CONTA1
OUT MEM10

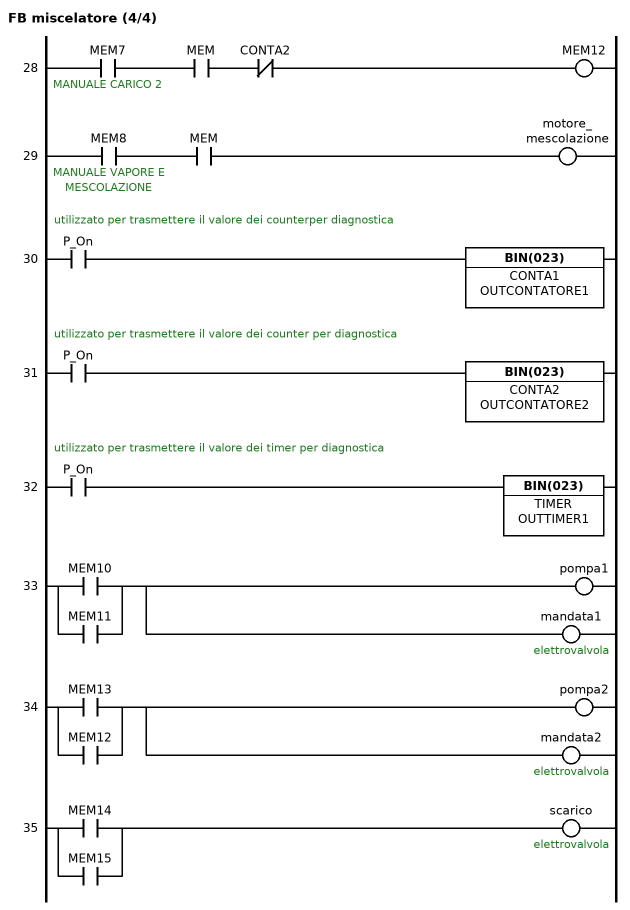
; rung 28
LD MEM7  ; MANUALE CARICO 2
AND MEM
ANDNOT CONTA2
OUT MEM12
; rung 29
LD MEM8  ; MANUALE VAPORE E MESCOLAZIONE
AND MEM
OUT motore_mescolazione
; rung 30: utilizzato per trasmettere il valore dei counterper diagnostica
LD P_On
BIN(023) CONTA1 OUTCONTATORE1
; rung 31: utilizzato per trasmettere il valore dei counter per diagnostica
LD P_On
BIN(023) CONTA2 OUTCONTATORE2
; rung 32: utilizzato per trasmettere il valore dei timer per diagnostica
LD P_On
BIN(023) TIMER OUTTIMER1
; rung 33
LD MEM10
OR MEM11
OUT pompa1
OUT mandata1  ; elettrovalvola
; rung 34
LD MEM13
OR MEM12
OUT pompa2
OUT mandata2  ; elettrovalvola
; rung 35
LD MEM14
OR MEM15
OUT scarico  ; elettrovalvola

## Function block semaforo_pedonale
VAR_INPUT
  pedonale1 : BOOL;
  pedonale2 : BOOL;
END_VAR
VAR_OUTPUT
  verde_pedoni : BOOL;
  rosso_pedoni : BOOL;
  verde_auto : BOOL;
  giallo_auto : BOOL;
  rosso_auto : BOOL;
  OUT_TIMER1 : WORD;
  OUT_TIMER2 : WORD;
  OUT_TIMER3 : WORD;
  OUT_TIMER4 : WORD;
  OUT_TIMER5 : WORD;
END_VAR
VAR
  MEM1 : BOOL;
  TIMER1 : TIMER;
  TIMER5 : TIMER;
  TIMER4 : TIMER;
  TIMER3 : TIMER;
  TIMER2 : TIMER;
END_VAR

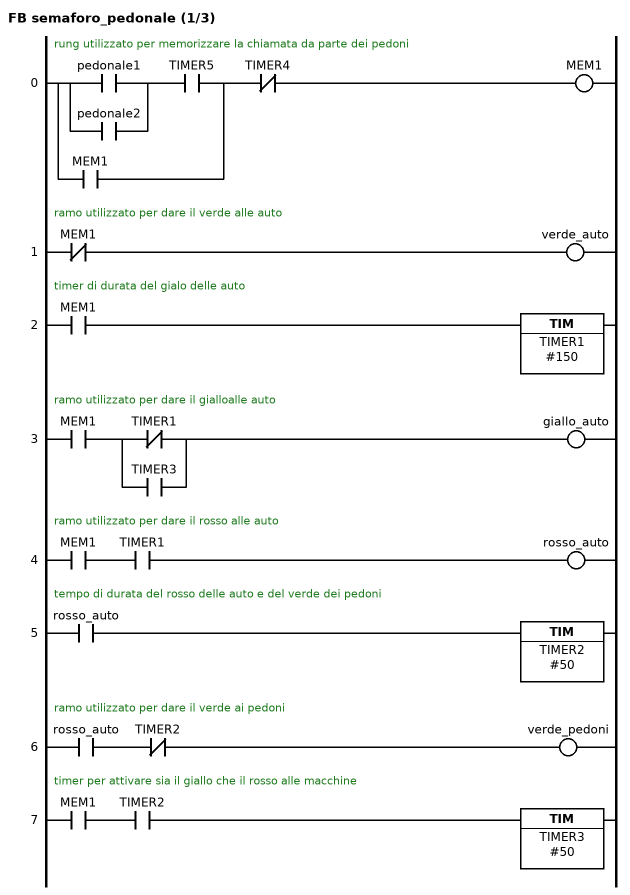
; rung 0: rung utilizzato per memorizzare la chiamata da parte dei pedoni
LD pedonale1
OR pedonale2
AND TIMER5
OR MEM1
ANDNOT TIMER4
OUT MEM1
; rung 1: ramo utilizzato per dare il verde alle auto
LDNOT MEM1
OUT verde_auto
; rung 2: timer di durata del gialo delle auto
LD MEM1
TIM TIMER1 #150
; rung 3: ramo utilizzato per dare il gialloalle auto
LD MEM1
LDNOT TIMER1
OR TIMER3
ANDLD
OUT giallo_auto
; rung 4: ramo utilizzato per dare il rosso alle auto
LD MEM1
AND TIMER1
OUT rosso_auto
; rung 5: tempo di durata del rosso delle auto e del verde dei pedoni
LD rosso_auto
TIM TIMER2 #50
; rung 6: ramo utilizzato per dare il verde ai pedoni
LD rosso_auto
ANDNOT TIMER2
OUT verde_pedoni
; rung 7: timer per attivare sia il giallo che il rosso alle macchine
LD MEM1
AND TIMER2
TIM TIMER3 #50

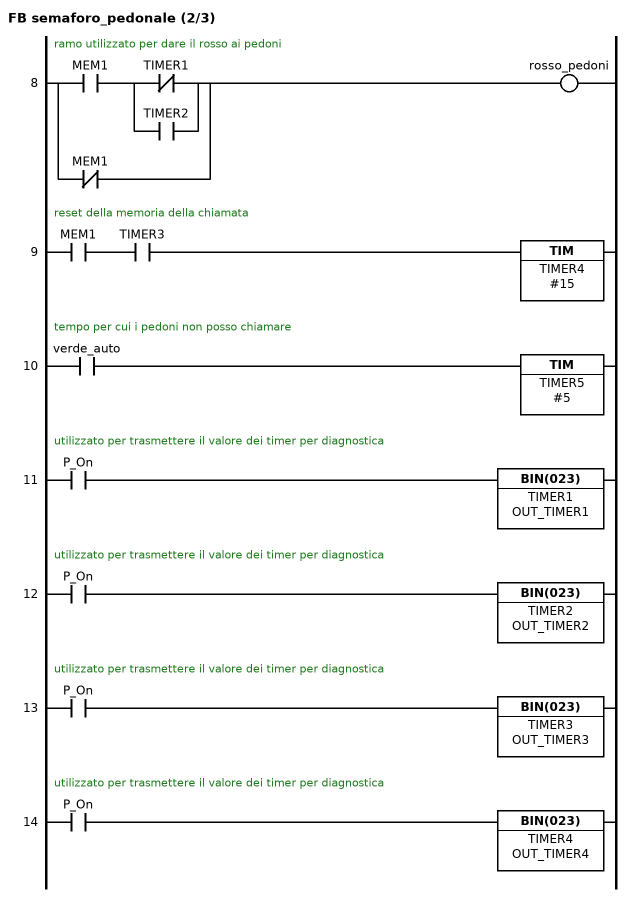
; rung 8: ramo utilizzato per dare il rosso ai pedoni
LD MEM1
LDNOT TIMER1
OR TIMER2
ANDLD
ORNOT MEM1
OUT rosso_pedoni
; rung 9: reset della memoria della chiamata
LD MEM1
AND TIMER3
TIM TIMER4 #15
; rung 10: tempo per cui i pedoni non posso chiamare
LD verde_auto
TIM TIMER5 #5
; rung 11: utilizzato per trasmettere il valore dei timer per diagnostica
LD P_On
BIN(023) TIMER1 OUT_TIMER1
; rung 12: utilizzato per trasmettere il valore dei timer per diagnostica
LD P_On
BIN(023) TIMER2 OUT_TIMER2
; rung 13: utilizzato per trasmettere il valore dei timer per diagnostica
LD P_On
BIN(023) TIMER3 OUT_TIMER3
; rung 14: utilizzato per trasmettere il valore dei timer per diagnostica
LD P_On
BIN(023) TIMER4 OUT_TIMER4

